Staubli VAL3: getTravelDist.pgx

program getTravelDist(num x_nIdx (dimensions=1), num& x_nTravelDist[] (dimensions=1), num& x_nError[] (dimensions=1))
  local num l_nEncValue
begin
  // This program returns the distance between the instantaneous
  // conveyor's position and the one when it was last latched.
  //
  // Input param
  //  x_nIdx    : Index of the object in the queue
  //
  // Output param
  //  x_nTravelDist : Distance
  //  x_nError      : Error code
  //    0 : No error
  //    1 : No object available
  //
  //----------------------------------------------------------------
  //
  x_nError=0
  if nNumbOfUser[x_nIdx]!=0
    l_nEncValue=aioGet(enc:aiEncCurrentPos)
    // Test for encoder roll over
    if l_nEncValue<nEncLatchedVal[x_nIdx]
      // roll over
      x_nTravelDist=nENCSCALEFACTOR*(enc:nMAXCOUNT-nEncLatchedVal[x_nIdx]+l_nEncValue-enc:nMINCOUNT)
    else
      // No roll over
      x_nTravelDist=nENCSCALEFACTOR*(l_nEncValue-nEncLatchedVal[x_nIdx])
    endIf
  else
    //* No Object requested
    x_nError=1
    if cfg:bLog==true
      nErrVal[0]=x_nIdx
      call ut:addNumToString(sConvNum+"(getTravelDist)>>:"+sErrMsgList[x_nError],sMsg,"*",nErrVal)
      logMsg(sMsg)
    endIf
  endIf
end
